{attribute addProperty BoxType "KL6581-0002"}
{attribute addProperty Id "Channel_1Channel_63387A5900"}
{attribute addProperty CRC "4090938439"}
{attribute addProperty SizeInBites "0"}
{attribute addProperty SizeInBytes "0"}
TYPE KL_F3D6C447 :
STRUCT
	{attribute addProperty Name "Channel_1"}
	Channel_1 : Channel_63387A59;
END_STRUCT
END_TYPE

(* stored: Version 1.2.0.0, ProductVersion 3.1.4024.9
   DUT KL_F3D6C447: Id {d7a65561-3864-4025-a878-82ae8410fa88} *)
